(* PLC project Unnamed, Unknown Unnamed 1 *)
(* stored: creationDateTime 2026-08-16T14:58:07, modificationDateTime 2026-08-16T14:58:07 *)

FUNCTION_BLOCK CTU
  VAR_OUTPUT
    Q : BOOL;
    CV : INT;
  END_VAR
  VAR_INPUT
    CU : BOOL;
    R : BOOL;
    PV : INT;
  END_VAR

END_FUNCTION_BLOCK

FUNCTION GE : BOOL
  VAR_INPUT
    IN1 : ANY_ELEMENTARY;
    IN2 : ANY_ELEMENTARY;
  END_VAR

END_FUNCTION

FUNCTION LE : BOOL
  VAR_INPUT
    IN1 : ANY_ELEMENTARY;
    IN2 : ANY_ELEMENTARY;
  END_VAR

END_FUNCTION

FUNCTION_BLOCK R_TRIG
  VAR_OUTPUT
    Q : BOOL;
  END_VAR
  VAR_INPUT
    CLK : BOOL;
  END_VAR

END_FUNCTION_BLOCK

FUNCTION_BLOCK SR
  VAR_OUTPUT
    Q1 : BOOL;
  END_VAR
  VAR_INPUT
    S1 : BOOL;
    R : BOOL;
  END_VAR

END_FUNCTION_BLOCK

FUNCTION_BLOCK TON
  VAR_OUTPUT
    Q : BOOL;
    ET : TIME;
  END_VAR
  VAR_INPUT
    IN : BOOL;
    PT : TIME;
  END_VAR

END_FUNCTION_BLOCK

PROGRAM automated_conveyor_checkweigher_and_batching_system
  VAR
    START_PB AT %IX0.0 : BOOL := FALSE;  (* START BUTTON *)
    STOP_PB AT %IX0.1 : BOOL := FALSE;  (* STOP BUTTON *)
    ESTOP_OK AT %IX0.2 : BOOL := TRUE;  (* E-STOP HEALTHY *)
    OVRLOAD_OK AT %IX0.3 : BOOL := TRUE;  (* OVERLOAD HEALTHY *)
    MOTOR_RUN AT %QX0.0 : BOOL;  (* MOTOR OUTPUT *)
    LAMP_RUN AT %QX0.1 : BOOL;  (* RUNNING INDICATOR *)
    PRODUCT_SENSOR AT %IX0.4 : BOOL := FALSE;  (* DETECTING PRODUCTS *)
    REJECT_SELENOID AT %QX0.2 : BOOL := FALSE;
  END_VAR
  VAR
    TON0 : TON;
    REJECT_PENDING : BOOL;
    SR0 : SR;
    TON1 : TON;
    REJECT_RESET : BOOL := FALSE;
    R_TRIG0 : R_TRIG;
    TON2 : TON;
    QUALITY_SENSOR : BOOL;
    R_TRIG1 : R_TRIG;
    BATCH_RESET_PB : BOOL;
    BATCH_COMPLETE_LAMP : BOOL;
    CTU1 : CTU;
    TON3 : TON;
    TON4 : TON;
    RAW_WEIGHT : INT := 0;  (* Raw integer reading from the scale's analog channel(0 - 32767) *)
    RAW_REAL : REAL := 0.0;  (* Temporary Floating_point values for maths *)
    SCALE_FACTOR : REAL := 0.00152588;  (* Coversion multiplier max kg/max raw = 50.0/32767.0 *)
    ACTUAL_WEIGHT : REAL := 0.0;  (* Calculated real weight of the product in kgs *)
    MIN_WEIGHT : REAL := 49.95;  (* Lower allowed limit *)
    MAX_WEIGHT : REAL := 50.10;  (* Upper allowed limit *)
    WEIGHT_OK : BOOL := FALSE;  (* Internal flag: TRUE when weight is valid *)
    ABOVE_MIN : BOOL;
    BELOW_MAX : BOOL;
  END_VAR
  VAR  (* added by the conversion: wires and edge detectors of the diagram *)
    _GE10858314_ENO : BOOL;
    _GE10858314_OUT : BOOL;
    _LE5869513_ENO : BOOL;
    _LE5869513_OUT : BOOL;
  END_VAR

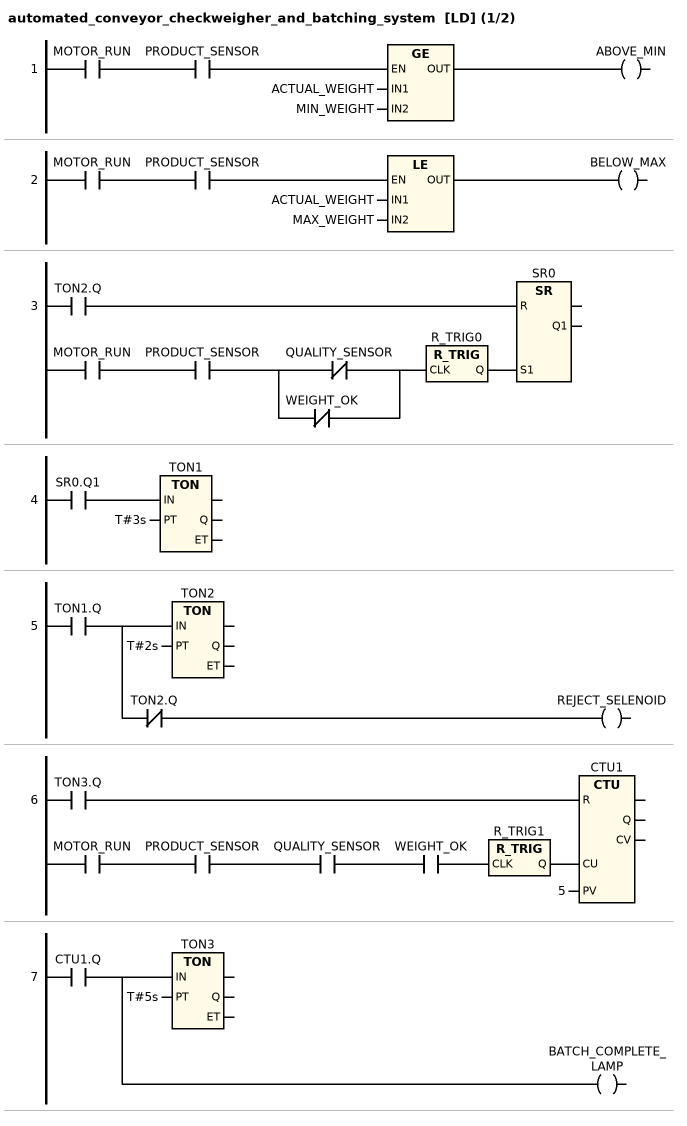
(* LD diagram, written out as Structured Text *)
MOTOR_RUN := NOT STOP_PB AND ESTOP_OK AND OVRLOAD_OK AND (START_PB OR MOTOR_RUN);
LAMP_RUN := MOTOR_RUN;
_GE10858314_OUT := GE(EN := MOTOR_RUN AND PRODUCT_SENSOR, IN1 := ACTUAL_WEIGHT, IN2 := MIN_WEIGHT, ENO => _GE10858314_ENO);
ABOVE_MIN := _GE10858314_OUT;
_LE5869513_OUT := LE(EN := MOTOR_RUN AND PRODUCT_SENSOR, IN1 := ACTUAL_WEIGHT, IN2 := MAX_WEIGHT, ENO => _LE5869513_ENO);
BELOW_MAX := _LE5869513_OUT;
WEIGHT_OK := MOTOR_RUN AND PRODUCT_SENSOR AND ABOVE_MIN AND BELOW_MAX;
REJECT_SELENOID := TON1.Q AND NOT TON2.Q;
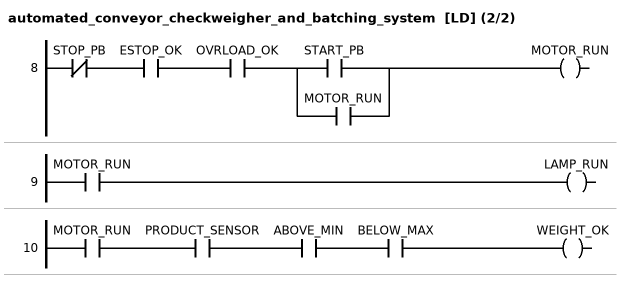
BATCH_COMPLETE_LAMP := CTU1.Q;
TON1(IN := SR0.Q1, PT := T#3s);
 := TON1.ET;
TON2(IN := TON1.Q, PT := T#2s);
 := TON2.ET;
R_TRIG1(CLK := MOTOR_RUN AND PRODUCT_SENSOR AND QUALITY_SENSOR AND WEIGHT_OK);
CTU1(CU := R_TRIG1.Q, R := TON3.Q, PV := 5);
 := CTU1.CV;
TON3(IN := CTU1.Q, PT := T#5s);
 := TON3.ET;
R_TRIG0(CLK := MOTOR_RUN AND PRODUCT_SENSOR AND (NOT QUALITY_SENSOR OR NOT WEIGHT_OK));
SR0(S1 := R_TRIG0.Q, R := TON2.Q);
END_PROGRAM

CONFIGURATION Config0
  RESOURCE Res0 ON PLC
    TASK task1(INTERVAL := T#20ms, PRIORITY := 1);
    PROGRAM instance1 WITH task1 : automated_conveyor_checkweigher_and_batching_system;
  END_RESOURCE
END_CONFIGURATION
